% RSLogix 500 project INTRO TO PLC - JOB 23.RSS, saved by version 10.00.00.00 %
PROJECT "PL06B"    % processor: Bul.1763 MicroLogix 1100 Series B %

PROGRAM FILES
  LAD 2   20 rungs

DATA FILES
  O0 OUTPUT  4 elements
  I1 INPUT  6 elements
  S2 STATUS  66 elements
  B3 BINARY  1 elements
  T4 TIMER  10 elements
  C5 COUNTER  3 elements
  R6 CONTROL  1 elements
  N7 INTEGER  5 elements
  F8 FLOAT  1 elements

LADDER 2
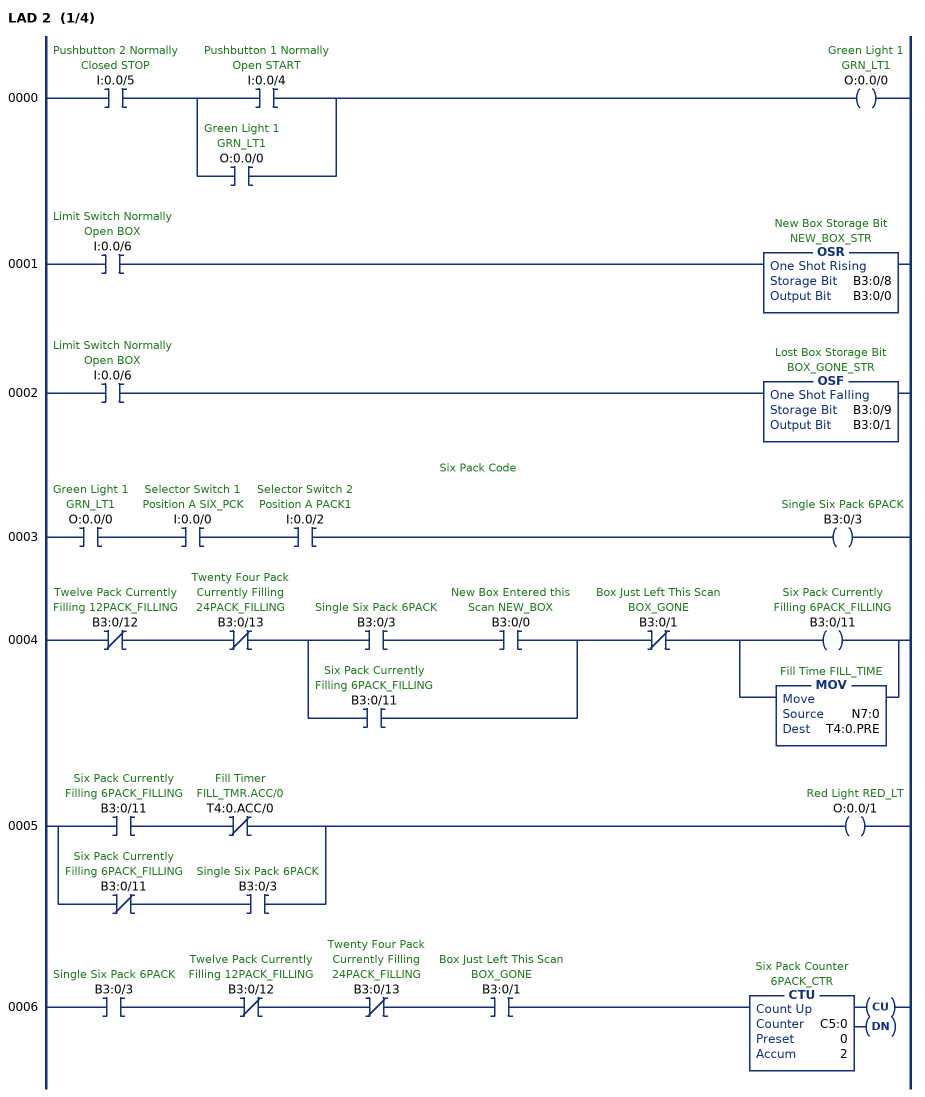
% Rung: 0 %
SOR XIC I:0.0/5 BST XIC I:0.0/4 NXB XIC O:0.0/0 BND OTE O:0.0/0 EOR
%   I:0.0/5  STOP  "Pushbutton 2 Normally Closed" %
%   I:0.0/4  START  "Pushbutton 1 Normally Open" %
%   O:0.0/0  GRN_LT1  "Green Light 1" %
% Rung: 1 %
SOR XIC I:0.0/6 OSR B3:0/8 B3:0/0 EOR
%   I:0.0/6  BOX  "Limit Switch Normally Open" %
%   B3:0/8  NEW_BOX_STR  "New Box Storage Bit" %
%   B3:0/0  NEW_BOX  "New Box Entered this Scan" %
% Rung: 2 %
SOR XIC I:0.0/6 OSF B3:0/9 B3:0/1 EOR
%   I:0.0/6  BOX  "Limit Switch Normally Open" %
%   B3:0/9  BOX_GONE_STR  "Lost Box Storage Bit" %
%   B3:0/1  BOX_GONE  "Box Just Left This Scan" %
% Rung: 3 %
% Six Pack Code %
SOR XIC O:0.0/0 XIC I:0.0/0 XIC I:0.0/2 OTE B3:0/3 EOR
%   O:0.0/0  GRN_LT1  "Green Light 1" %
%   I:0.0/0  SIX_PCK  "Selector Switch 1 Position A" %
%   I:0.0/2  PACK1  "Selector Switch 2 Position A" %
%   B3:0/3  6PACK  "Single Six Pack" %
% Rung: 4 %
SOR XIO B3:0/12 XIO B3:0/13 BST XIC B3:0/3 XIC B3:0/0 NXB XIC B3:0/11 BND XIO B3:0/1 BST OTE B3:0/11 NXB MOV N7:0 T4:0.PRE BND EOR
%   B3:0/12  12PACK_FILLING  "Twelve Pack Currently Filling" %
%   B3:0/13  24PACK_FILLING  "Twenty Four Pack Currently Filling" %
%   B3:0/3  6PACK  "Single Six Pack" %
%   B3:0/0  NEW_BOX  "New Box Entered this Scan" %
%   B3:0/11  6PACK_FILLING  "Six Pack Currently Filling" %
%   B3:0/1  BOX_GONE  "Box Just Left This Scan" %
%   N7:0  6PACK_FILL_TIME  "Six Pack Fill Time" %
%   T4:0.PRE  FILL_TIME  "Fill Time" %
% Rung: 5 %
SOR BST XIC B3:0/11 XIO T4:0.ACC/0 NXB XIO B3:0/11 XIC B3:0/3 BND OTE O:0.0/1 EOR
%   B3:0/11  6PACK_FILLING  "Six Pack Currently Filling" %
%   T4:0  FILL_TMR  "Fill Timer" %
%   B3:0/3  6PACK  "Single Six Pack" %
%   O:0.0/1  RED_LT  "Red Light" %
% Rung: 6 %
SOR XIC B3:0/3 XIO B3:0/12 XIO B3:0/13 XIC B3:0/1 CTU C5:0 0 2 EOR
%   B3:0/3  6PACK  "Single Six Pack" %
%   B3:0/12  12PACK_FILLING  "Twelve Pack Currently Filling" %
%   B3:0/13  24PACK_FILLING  "Twenty Four Pack Currently Filling" %
%   B3:0/1  BOX_GONE  "Box Just Left This Scan" %
%   C5:0  6PACK_CTR  "Six Pack Counter" %

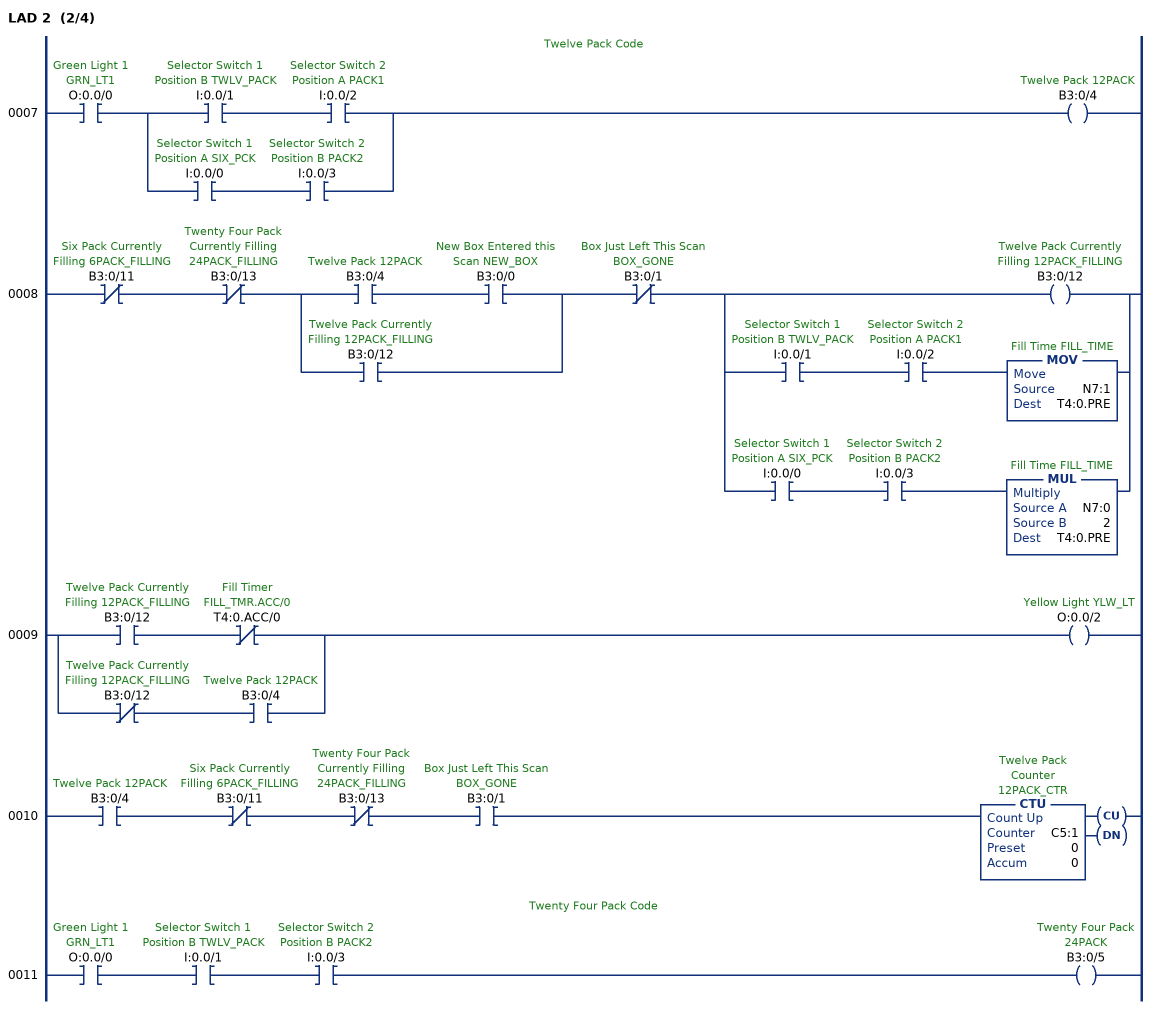
% Rung: 7 %
% Twelve Pack Code %
SOR XIC O:0.0/0 BST XIC I:0.0/1 XIC I:0.0/2 NXB XIC I:0.0/0 XIC I:0.0/3 BND OTE B3:0/4 EOR
%   O:0.0/0  GRN_LT1  "Green Light 1" %
%   I:0.0/1  TWLV_PACK  "Selector Switch 1 Position B" %
%   I:0.0/2  PACK1  "Selector Switch 2 Position A" %
%   I:0.0/0  SIX_PCK  "Selector Switch 1 Position A" %
%   I:0.0/3  PACK2  "Selector Switch 2 Position B" %
%   B3:0/4  12PACK  "Twelve Pack" %
% Rung: 8 %
SOR XIO B3:0/11 XIO B3:0/13 BST XIC B3:0/4 XIC B3:0/0 NXB XIC B3:0/12 BND XIO B3:0/1 BST OTE B3:0/12 NXB XIC I:0.0/1 XIC I:0.0/2 MOV N7:1 T4:0.PRE NXB XIC I:0.0/0 XIC I:0.0/3 MUL N7:0 2 T4:0.PRE BND EOR
%   B3:0/11  6PACK_FILLING  "Six Pack Currently Filling" %
%   B3:0/13  24PACK_FILLING  "Twenty Four Pack Currently Filling" %
%   B3:0/4  12PACK  "Twelve Pack" %
%   B3:0/0  NEW_BOX  "New Box Entered this Scan" %
%   B3:0/12  12PACK_FILLING  "Twelve Pack Currently Filling" %
%   B3:0/1  BOX_GONE  "Box Just Left This Scan" %
%   I:0.0/1  TWLV_PACK  "Selector Switch 1 Position B" %
%   I:0.0/2  PACK1  "Selector Switch 2 Position A" %
%   N7:1  12PACK_FILL_TIME  "Twelve Pack Fill Time" %
%   T4:0.PRE  FILL_TIME  "Fill Time" %
%   I:0.0/0  SIX_PCK  "Selector Switch 1 Position A" %
%   I:0.0/3  PACK2  "Selector Switch 2 Position B" %
%   N7:0  6PACK_FILL_TIME  "Six Pack Fill Time" %
% Rung: 9 %
SOR BST XIC B3:0/12 XIO T4:0.ACC/0 NXB XIO B3:0/12 XIC B3:0/4 BND OTE O:0.0/2 EOR
%   B3:0/12  12PACK_FILLING  "Twelve Pack Currently Filling" %
%   T4:0  FILL_TMR  "Fill Timer" %
%   B3:0/4  12PACK  "Twelve Pack" %
%   O:0.0/2  YLW_LT  "Yellow Light" %
% Rung: 10 %
SOR XIC B3:0/4 XIO B3:0/11 XIO B3:0/13 XIC B3:0/1 CTU C5:1 0 0 EOR
%   B3:0/4  12PACK  "Twelve Pack" %
%   B3:0/11  6PACK_FILLING  "Six Pack Currently Filling" %
%   B3:0/13  24PACK_FILLING  "Twenty Four Pack Currently Filling" %
%   B3:0/1  BOX_GONE  "Box Just Left This Scan" %
%   C5:1  12PACK_CTR  "Twelve Pack Counter" %
% Rung: 11 %
% Twenty Four Pack Code %
SOR XIC O:0.0/0 XIC I:0.0/1 XIC I:0.0/3 OTE B3:0/5 EOR
%   O:0.0/0  GRN_LT1  "Green Light 1" %
%   I:0.0/1  TWLV_PACK  "Selector Switch 1 Position B" %
%   I:0.0/3  PACK2  "Selector Switch 2 Position B" %
%   B3:0/5  24PACK  "Twenty Four Pack" %

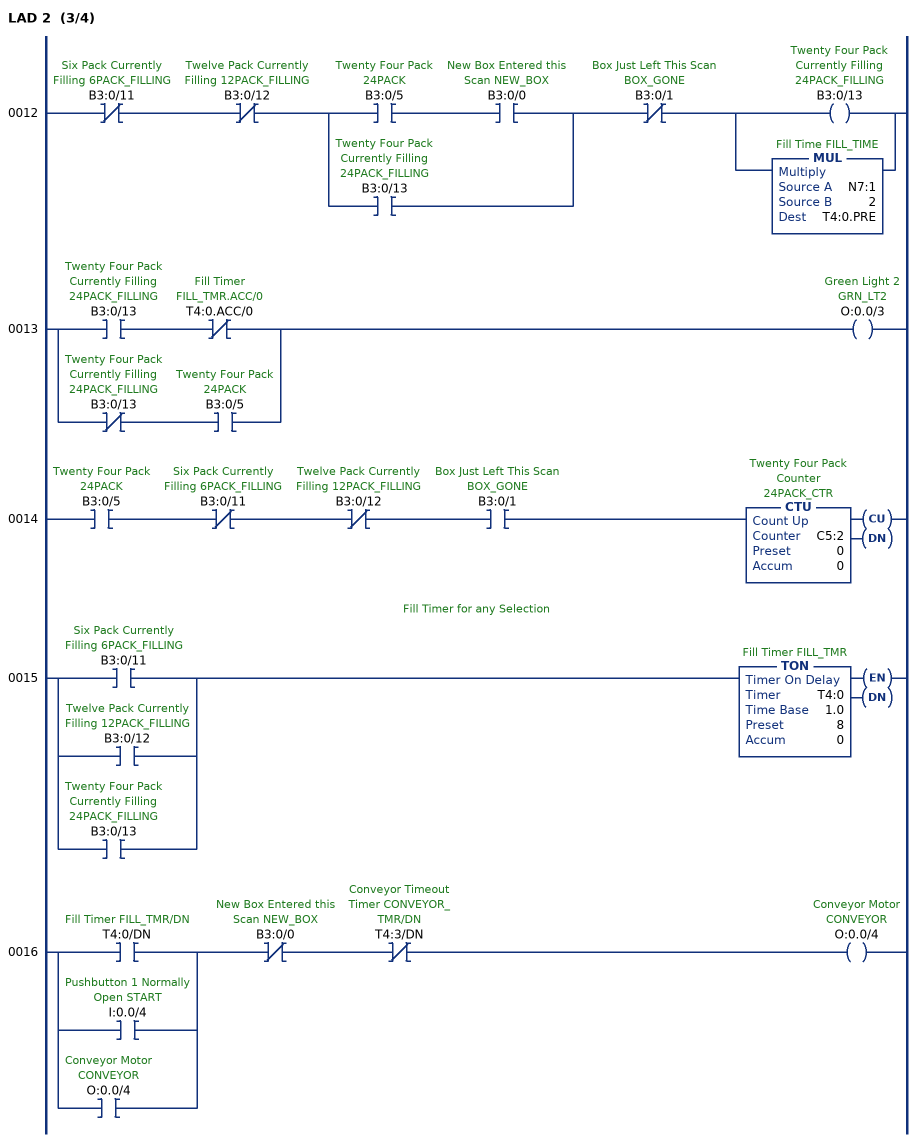
% Rung: 12 %
SOR XIO B3:0/11 XIO B3:0/12 BST XIC B3:0/5 XIC B3:0/0 NXB XIC B3:0/13 BND XIO B3:0/1 BST OTE B3:0/13 NXB MUL N7:1 2 T4:0.PRE BND EOR
%   B3:0/11  6PACK_FILLING  "Six Pack Currently Filling" %
%   B3:0/12  12PACK_FILLING  "Twelve Pack Currently Filling" %
%   B3:0/5  24PACK  "Twenty Four Pack" %
%   B3:0/0  NEW_BOX  "New Box Entered this Scan" %
%   B3:0/13  24PACK_FILLING  "Twenty Four Pack Currently Filling" %
%   B3:0/1  BOX_GONE  "Box Just Left This Scan" %
%   N7:1  12PACK_FILL_TIME  "Twelve Pack Fill Time" %
%   T4:0.PRE  FILL_TIME  "Fill Time" %
% Rung: 13 %
SOR BST XIC B3:0/13 XIO T4:0.ACC/0 NXB XIO B3:0/13 XIC B3:0/5 BND OTE O:0.0/3 EOR
%   B3:0/13  24PACK_FILLING  "Twenty Four Pack Currently Filling" %
%   T4:0  FILL_TMR  "Fill Timer" %
%   B3:0/5  24PACK  "Twenty Four Pack" %
%   O:0.0/3  GRN_LT2  "Green Light 2" %
% Rung: 14 %
SOR XIC B3:0/5 XIO B3:0/11 XIO B3:0/12 XIC B3:0/1 CTU C5:2 0 0 EOR
%   B3:0/5  24PACK  "Twenty Four Pack" %
%   B3:0/11  6PACK_FILLING  "Six Pack Currently Filling" %
%   B3:0/12  12PACK_FILLING  "Twelve Pack Currently Filling" %
%   B3:0/1  BOX_GONE  "Box Just Left This Scan" %
%   C5:2  24PACK_CTR  "Twenty Four Pack Counter" %
% Rung: 15 %
% Fill Timer for any Selection %
SOR BST XIC B3:0/11 NXB XIC B3:0/12 NXB XIC B3:0/13 BND TON T4:0 1.0 8 0 EOR
%   B3:0/11  6PACK_FILLING  "Six Pack Currently Filling" %
%   B3:0/12  12PACK_FILLING  "Twelve Pack Currently Filling" %
%   B3:0/13  24PACK_FILLING  "Twenty Four Pack Currently Filling" %
%   T4:0  FILL_TMR  "Fill Timer" %
% Rung: 16 %
SOR BST XIC T4:0/DN NXB XIC I:0.0/4 NXB XIC O:0.0/4 BND XIO B3:0/0 XIO T4:3/DN OTE O:0.0/4 EOR
%   T4:0  FILL_TMR  "Fill Timer" %
%   I:0.0/4  START  "Pushbutton 1 Normally Open" %
%   O:0.0/4  CONVEYOR  "Conveyor Motor" %
%   B3:0/0  NEW_BOX  "New Box Entered this Scan" %
%   T4:3  CONVEYOR_TMR  "Conveyor Timeout Timer" %

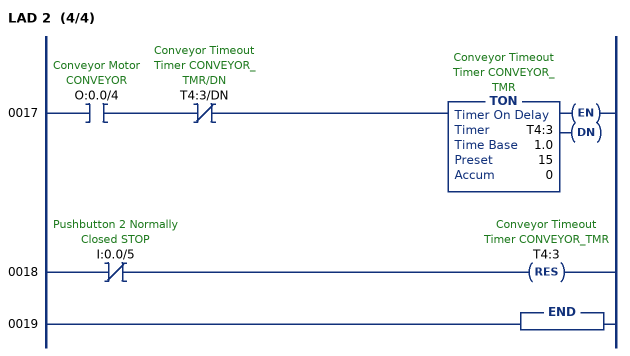
% Rung: 17 %
SOR XIC O:0.0/4 XIO T4:3/DN TON T4:3 1.0 15 0 EOR
%   O:0.0/4  CONVEYOR  "Conveyor Motor" %
%   T4:3  CONVEYOR_TMR  "Conveyor Timeout Timer" %
% Rung: 18 %
SOR XIO I:0.0/5 RES T4:3 EOR
%   I:0.0/5  STOP  "Pushbutton 2 Normally Closed" %
%   T4:3  CONVEYOR_TMR  "Conveyor Timeout Timer" %
% Rung: 19 %
SOR END EOR

OTHER DOCUMENTED ADDRESSES
  B3:0/6  2TWLVPACK  "Two Twelve Packs"
  B3:0/15  SCRATCH  "Scratch Bit"
  B3:1/1  RED_TMR_DNS  "New Box"
  I  
  RTC:0.YR  RTC
  SEL1B  
  T4:1  12PACK_TMR  "Two Six Pack Timer"
  T4:2  24PACK_TMR  "Twelve Pack Timer"

DATA TABLE (non-zero values as saved)
DATA B3
% B3:0 % 0X8008
DATA T4
% .PRE .ACC %
% T4:0 % 8 0
% T4:2 % 13 0
% T4:3 % 15 0
DATA C5
% .PRE .ACC %
% C5:0 % 0 2
DATA N7
% N7:0 % 8 13 0 0 0
